FUNCTION F_TrackSettingChangesB : BOOL
VAR_INPUT
	bValue		: BOOL;
END_VAR
VAR_IN_OUT
	stSetting	: ST_Data_Item;
	sChanges	: STRING;
END_VAR

IF stSetting.bValue <> bValue THEN
	sChanges := Concat7(sChanges, '$N ', WSTRING_TO_STRING(stSetting.stName.wsName), ' ', TO_STRING(stSetting.bValue), ' -> ', TO_STRING(bValue));
END_IF

stSetting.bValue := bValue;
F_TrackSettingChangesB := TRUE;

END_FUNCTION

(* stored: Version 1.1.0.1, ProductVersion 3.1.4024.12
   POU F_TrackSettingChangesB: Id {836ae16d-cbe0-4b90-9ab5-901d5f8fb1e3}, SpecialFunc None *)
